TYPE ST_PROCESS_DATA :
STRUCT
  ActiveStations      : T_PROCESS; // where and how many stations are to be used in process
  ProcessTarget       : UINT;      // for whom?
END_STRUCT
END_TYPE

(* stored: Version 1.1.0.1
   DUT ST_PROCESS_DATA: Id {07616521-f21e-48a7-acef-db6b7d7585de} *)
